METHOD PROTECTED ExecFaultHandling : BOOL
VAR
	bEnableCheck: BOOL ; // enable check functions 
	nActPos		: LREAL; // actual position of traverse axis (for readability)	 
	bActMovFwd	: BOOL ; // traverse is moving in positive direction
	bActMovRev	: BOOL ; // traverse is moving in negative direction
END_VAR
// ====== Write axis position to temporary variable to improver readability =======
	nActPos := stTraverseAxisRef.NcToPlc.ActPos ;
	IF stTraverseAxisRef.Status.Moving THEN 
		bActMovFwd := stTraverseAxisRef.Status.PositiveDirection ; 
		bActMovRev := stTraverseAxisRef.Status.NegativeDirection ; 
	ELSE
		bActMovFwd := FALSE ; 
		bActMovRev := FALSE ; 
	END_IF
	
// ====== Alway check if cylinder is down when within minimum range ======
	fbTimerStartup(IN := NOT bErrorActive, PT := LREAL_TO_TIME(stParTimeToClose.fValue));
	
	IF fbTimerStartup.Q 
	AND	nActPos > nTriggerPosUprev 
	AND nActPos < nTriggerPosUpFw 
	AND NOT fbSensorClosed.bFcoInputActive  THEN 	
		// Set error to active (stop traverse axis) 
		bErrorActive := TRUE ;
		// add message data
		stFault.Active			:= TRUE 								;
		stFault.Discription		:= 'support not in safe (down) position';
		stFault.MessageNumber	:= E_MessageNumbers.FF_Collision 		;
		stFault.FaultType		:= E_FaultTypes.FF				;
		refFbFault.CmdAddFault( stFault );
	END_IF

// ====== Make sure support Moves down ======
	IF bActMovFwd 
	AND nActPos > nTriggerPosCheckDownFw 
	AND nActPos < nTriggerPosUpFw 
	AND NOT fbSensorClosed.bFcoInputActive THEN 
		// Set error to active (stop traverse axis) 
		bErrorActive := TRUE ;
		// add message data
		stFault.Active			:= TRUE 								;
		stFault.Discription		:= 'Emergency stop support cylinder not down';
		stFault.MessageNumber	:= E_MessageNumbers.FF_Collision 		;
		stFault.FaultType		:= E_FaultTypes.FF				;
		refFbFault.CmdAddFault( stFault );
	ELSIF bActMovRev 
	AND nActPos > nTriggerPosUprev
	AND nActPos < nTriggerPosCheckDownRe 
	AND NOT fbSensorClosed.bFcoInputActive THEN 
		// Set error to active (stop traverse axis) 
		bErrorActive := TRUE ;
		// add message data
		stFault.Active			:= TRUE 								;
		stFault.Discription		:= 'Emergency stop support cylinder not down';
		stFault.MessageNumber	:= E_MessageNumbers.FF_Collision 		;
		stFault.FaultType		:= E_FaultTypes.FF				;
		refFbFault.CmdAddFault( stFault );
 	END_IF
END_METHOD

METHOD Init_Support : BOOL
VAR_INPUT
	sInValveName		: STRING			:= 'valve'	; // Name of the cylinder ( used for fault handling and identification)
	nInValveNumber		: UDINT				:= 0		; // Cylinder identification number
	// Support data
	nInSupportPosition	: LREAL := 0 		; // possition of support cylinder in reference to the home position 
	nInSupportWidth		: LREAL := 100		; // width of support cylinder 
	// Traverse data 
	nInTravMaxAcc			: LREAL ; // traverse maximum acceleration 
	nInTravMaxDec			: LREAL ; // traverse maximum deceleration 
	nInTraverseLength		: LREAL	:= 550		; // Length of sewing head cart 
	nInTraverseFlagPosition	: LREAL	:= 0		; // position of flag in reference to edge of cart 
	// cart data
	nInHandCartLenght		: LREAL := 250		; // hand cart length [mm]
	nInHandCartClearance	: LREAL := 300		; // Clearance around cart in which support is down

	// safety values 	
	nInMinSafeDistanceDown: LREAL := 200		; // Minimum distance for support to move down
	// Command state
	eResetState		: E_ValveResetState := 0		; // Cylinder reset state variable (default is idle) 
	eSafeState		: E_ValveResetState	:= 0		; // Valve safe state
END_VAR
// ====== initi valve ======
	SUPER^.Init(nInValveNumber, eResetState, eSafeState);
	
// ====== Set support data =======
	nSupportPosition 	:= nInSupportPosition 	;
	nSupportWidth		:= nInSupportWidth 		;

// ====== Set traverse Data ======
	nTravMaxAcc				:= nInTravMaxAcc			;
	nTravMaxDec				:= nInTravMaxDec			;
	nTraverseLength 		:= nInTraverseLength		;
	nTraverseFlagPosition	:= nInTraverseFlagPosition 	;
	nMinSafeDistanceDown	:= nInMinSafeDistanceDown	;

// ===== set handcart data =====
	nHandCartLength 		:= nInHandCartLenght 		;
	nHandCartClearance		:= nInHandCartClearance		;

// ====== set feedback to true (support always has feedback) =======
	bIcfFbkClosedPresent 	:= TRUE ;
	bIcfFbkOpenPresent		:= TRUE ;
	
// ====== Check if init is done ======
END_METHOD

METHOD PUBLIC Mod_ManualControl : BOOL
VAR_INPUT
	eCmdCylinder : E_CylinderCmd ; // cylinder manual command	
END_VAR
bCmdManual := TRUE ;

CASE eCmdCylinder OF
	E_CylinderCmd.Cyl_Reset:
		CmdReset();
	E_CylinderCmd.Cyl_Hold:
		CmdHold();
	E_CylinderCmd.Cyl_Teach:
		CmdTeach();
	E_CylinderCmd.Cyl_Calculate:
		ExecCalc();
	E_CylinderCmd.Cyl_Expand:
		CmdOpen();
	E_CylinderCmd.Cyl_Retract:
		CmdClose();
	ELSE 
		RETURN;
END_CASE
END_METHOD

METHOD Mod_SupportDown : BOOL
VAR_INPUT
END_VAR
bCmdSupportDown := true ;
END_METHOD

END_FUNCTION_BLOCK

// Axis/FunctionBlocks/FB_DevBasicACAxis
FUNCTION_BLOCK PUBLIC FB_DevBasicACAxis EXTENDS FB_DevBase
VAR_INPUT
	// ===== General Function input =====
		fCmdAcc			: LREAL := 15000;
		fCmdDecc		: LREAL := 15000; 
	// Manual control reference
		stManualCtrl	: UDT_ManualAxisCtrl ;
END_VAR
VAR_OUTPUT
	bHomed			: BOOL 	:= FALSE; 
	bMoving		: BOOL ; // Axis is moving
	bInPosition : BOOL ; // Axis is in position 
END_VAR
VAR
		AxisRef	: AXIS_REF ; // reference to AC axis
	// ===== HW Config Bits =====
		bIcfCmdVelocityRpm	: BOOL ; // input speeds in Rpm
		bIcfEnableForward 	: BOOL ; // Enable forward motion
 		bIcfEnablereverse	: BOOL ; // Enable reverse motion
		bIcfAlwaysEnable	: BOOL ; // 1 = Axis always enabled, 0 = Axis disabled at Idle 
		bIcfSimulationMode	: BOOL := FALSE ; // Simulation mode is active [default set to False] 
	// ===== Internal motion values ======
		fHomePosition		: LREAL := 0 ; // set position at homing
	// ====== Axis Settings ======
		fMaxVelo		: LREAL := 0 ; // Axis Maximum velocity
		fMaxAcc			: LREAL := 0 ; // Axis Maximum cceleration
		fMaxDec			: LREAL := 0 ; // axis Maxium deceleration 
		
		fSafeVeloLimit	: LREAL	:= 200; // Safe velocity limit 
		tEnableDelay	: TIME 	:= T#150MS	;
		tDisableDelay	: TIME 	:= T#500MS  ;
		
	// ====== Axis enable =====	
		bCmdEnableAxis 		: BOOL 	:= FALSE; // Command to enable the axis (External)
		bInternalEnable		: BOOL 	:= FALSE; // internal enable command (turns off after set time, and on at new motion command
		bDelayedEnable		: BOOL 	:= false; // Delayed enable signal for motion commands
		TonMotionEnable		: TON 			; // Timer on for motion command enable
		TofIntAxisEnable	: TOF  			; // Timer off for internal axis enable 
	// ===== Safe commands =====
		bCmdSafeStop	: BOOL ;
	// Motion commands 
		fbMcPower 			: MC_Power		;		// FB for enable and override
		fbMcReset 			: MC_Reset		;		// FB to reset axis
		fbSoeReset			: FB_SoEReset	; 		// FB to reset axis hardware
		fbMcHome			: MC_Home		;		// Fb to home Axis
		fbMcStop 			: MC_Stop		;		// FB to stop axis
		fbMcHalt			: MC_Halt		;		// FB to halt axis
		fbMcJog				: MC_Jog		;		// FB to Jog axis
		fbMcMoveVelocity	: MC_MoveVelocity;		// FB to move with specified velocity until Next command is given
	(* PtoP Motion move commands are in arrays so multiple commands can be stacked *) 
		fbMCMoveRelative	: ARRAY [0..1] OF MC_MoveRelative	;		// FB to move relative
		fbMcMoveAbsolute	: ARRAY [0..1] OF MC_MoveAbsolute	;		// FB to move axis (velocity movement)
		
	// Parameters 
		stMParMaxAcc : Udt_Parameter := (fMaximum := 999999, fMinimum := 0, fValue := 0)	; // Parameter for maximum acceleration
		stMParMaxDec : Udt_Parameter := (fMaximum := 999999, fMinimum := 0, fValue := 0)	; // Parameter for maximum Deceleration
		stMparMaxVelo: Udt_Parameter := (fMaximum := 999999, fMinimum := 0, fValue := 0)	; // Parameter for maximum velocity
		
	// Device feedback
		nActVelocity AT%I* : INT ; // actual speed of the motor
		nActPosition AT%I* : UDINT ; // Actual position of the motor

	// ===== Function execute triggers =====
		bExec_Reset			: BOOL := FALSE; // Execute reset
		bExec_Halt			: BOOL := FALSE; // Execute hold
		bExec_Home			: BOOL := FALSE; // Execute Home
		bExec_JogPositive	: BOOL := FALSE; // Execute Jog in positive direction
		bExec_JogNegative	: BOOL := FALSE; // Execute Jog in negative direction
		bExec_MoveVelocity	: BOOL := FALSE; // Execute move velocity
		arExec_MoveRelative	: ARRAY [0..1] OF BOOL ; // Execute move relative
		arExec_MoveAbs		: ARRAY [0..1] OF BOOL ; // Execute move absolute reverse
		

END_VAR

// Call base function
SUPER^(refFbFault := refFbFault);

// ==== Check if axis is initiated =====
IF NOT bInitOk THEN 
	RETURN ; 
END_IF

// ===== Execute safe functions =====
	ExecSafeFunctions(); 

// ==== Execute organizational functions =====
	ExecEnable();

// ==== execute motion functions =====
	CallMotionFunctions();

METHOD PUBLIC CmdHalt : BOOL
VAR_INPUT
	fDeceleration 	: LREAL := 0 ; // command deceleration
	mcBuffermode	: MC_BufferMode ; // Buffermode defines how the previous command is executed.
END_VAR
// Set command to true 
bExec_Halt 		:= TRUE ;
bInternalEnable	:= TRUE ;

// coppy parameters
fbMcHalt.Deceleration	:= fDeceleration;
fbMcHalt.BufferMode		:= mcBuffermode	;

// Set feedback output 
CmdHalt := fbMchalt.Active ;
END_METHOD

METHOD PUBLIC CmdHome : BOOL // start axis homing procedure
VAR_INPUT
	fPosition 		: LREAL := 0 ; // Homing position
	mcBufferMode	: MC_BufferMode := MC_BufferMode.MC_Aborting		; // Buffermode
END_VAR
// set command to true 
bExec_Home 		:= TRUE	; 
bInternalEnable	:= TRUE ;

// coppy parameters
fbMcHome.Position 	:= fPosition 	;
fbMcHome.BufferMode	:= mcBufferMode ;

// Set feedback output
CmdHome := fbMcHome.Done ;
END_METHOD

METHOD PUBLIC CmdJog : BOOL // Jog axis with variable speed. jog stops as soon as the command is false
VAR_INPUT
	fVelocity		: LREAL 	; // jog velocity can be adjusted as long as the command is active
	fPos			: LREAL 	; // Jog position or step size (if aplicable)
	bJogNegative 	: BOOL 		:= FALSE ; // jog in negative direction
	eJogmode		: E_JogMode := E_JogMode.MC_JOGMODE_CONTINOUS ; // jogmode [default MC_JOGMODE_CONTINOUS] 
END_VAR
// Velocity conversion from RPM to deg/sec
	IF bIcfCmdVelocityRpm THEN 
		fVelocity := Rpm_To_DegS(fVelocity);
	END_IF

// Set command to true
	IF fbMcJog.Velocity = fVelocity THEN // If command velocity changes, then set exec to false for one cycle to trigger new velocity so the jog follows the set velocity
		bExec_JogPositive	:= NOT bJogNegative ;
		bExec_JogNegative 	:= bJogNegative ;
	END_IF
	bInternalEnable			:= TRUE ;

// coppy parameters
	fbMcJog.Velocity	:= fVelocity 	;
	fbmcjog.Mode		:= eJogmode		;
	fbMcJog.Position	:= fPos			;

// Set feedback output 
	CmdJog := fbMcJog.Active ;
END_METHOD

METHOD PUBLIC CmdManual : BOOL
VAR
	eJogmode		: E_JogMode := E_JogMode.MC_JOGMODE_CONTINOUS ; // jogging mode 
END_VAR
// Enable axis for manual control
bCmdManual := TRUE ;

// set jog mode 
IF stManualCtrl.bCmdInching THEN 
	eJogmode := E_JogMode.MC_JOGMODE_INCHING ;
END_IF

// execute motion commands
IF stManualCtrl.bCmdJogForward OR stManualCtrl.bCmdJogReverse THEN 
	CmdJog (fVelocity := stManualCtrl.fVelocity, 
			fPos := stManualCtrl.fDistance, 
			bJogNegative := stManualCtrl.bCmdJogReverse, 
			eJogmode := eJogmode);
ELSIF stManualCtrl.bCmdToPos THEN 
	CmdMoveAbs( fPosition := stManualCtrl.fPosition, 
				fVelocity := stManualCtrl.fVelocity, 
				mcBuffermode := MC_BufferMode.MC_Aborting);
ELSIF stManualCtrl.bCmdHome THEN 
	CmdHome( fPosition := 0, mcBufferMode := MC_Aborting);
ELSE 
	CmdHalt( 	fDeceleration := fMaxDec * 0.9, 
				mcBuffermode := MC_BufferMode.MC_Aborting) ; 
END_IF
END_METHOD

METHOD PUBLIC CmdMoveAbs : BOOL // Move absolute command
VAR_INPUT
	fPosition	:	LREAL 	; // target position
	fVelocity	: 	LREAL 	; // Maximum velocity [units/sec]
	mcBuffermode: 	MC_BufferMode ; // Buffermode defines how the previous command is executed.
END_VAR
// Velocity conversion from RPM to deg/sec
	IF bIcfCmdVelocityRpm THEN 
		fVelocity := Rpm_To_DegS(fVelocity);
	END_IF

// Determine function for command stacking
	IF fbMcMoveAbsolute[0].Active THEN 
		arExec_MoveAbs[1] 				:= (fPosition <> fbMcMoveAbsolute[0].Position OR fVelocity <> fbMcMoveAbsolute[0].Velocity) ;
		fbMcMoveAbsolute[1].Position 	:= fPosition ;
		fbMcMoveAbsolute[1].Velocity 	:= fVelocity ; 
		fbMcMoveAbsolute[1].BufferMode 	:= mcBuffermode ;
	ELSE
		arExec_MoveAbs[0] 				:= (fPosition <> fbMcMoveAbsolute[1].Position OR fVelocity <> fbMcMoveAbsolute[1].Velocity) ;
		fbMcMoveAbsolute[0].Position 	:= fPosition ;
		fbMcMoveAbsolute[0].Velocity 	:= fVelocity ; 
		fbMcMoveAbsolute[0].BufferMode 	:= mcBuffermode ;
	END_IF

bInternalEnable	:= TRUE ;
// set feedback
IF arExec_MoveAbs[1] OR fbMcMoveAbsolute[1].Busy THEN 
	CmdMoveAbs :=	fbMcMoveAbsolute[1].Active ;
ELSE 
	CmdMoveAbs :=	fbMcMoveAbsolute[0].Active ;
END_IF
END_METHOD

METHOD CmdMoveRelative : BOOL // move relative command 
VAR_INPUT
	fDistance	:	LREAL 	; // target position
	fVelocity	: 	LREAL 	; // Maximum velocity [units/sec]
	mcBuffermode: 	MC_BufferMode ; // Buffermode defines how the previous command is executed.
END_VAR
// Velocity conversion from RPM to deg/sec
	IF bIcfCmdVelocityRpm THEN 
		fVelocity := Rpm_To_DegS(fVelocity);
	END_IF

// Determine function for command stacking
	IF fbMCMoveRelative[0].Active THEN 
		arExec_MoveRelative[1] := (fDistance <> fbMCMoveRelative[0].Distance OR fVelocity <> fbMCMoveRelative[0].Velocity) ;
		fbMCMoveRelative[1].Velocity	:= fVelocity 	;
		fbMCMoveRelative[1].Distance	:= fDistance	;
		fbMCMoveRelative[1].BufferMode	:= mcBuffermode	;
	ELSE 
		arExec_MoveRelative[0] := (fDistance <> fbMCMoveRelative[1].Distance OR fVelocity <> fbMCMoveRelative[1].Velocity) ;
		fbMCMoveRelative[0].Velocity	:= fVelocity 	;
		fbMCMoveRelative[0].Distance	:= fDistance	;
		fbMCMoveRelative[0].BufferMode	:= mcBuffermode	;
	END_IF

bInternalEnable	:= TRUE ;

// set feedback
IF arExec_MoveRelative[1] OR fbMCMoveRelative[1].Busy THEN 
	CmdMoveRelative :=	fbMCMoveRelative[1].Active ;
ELSE
	CmdMoveRelative :=	fbMCMoveRelative[0].Active ;
END_IF
END_METHOD

METHOD PUBLIC CmdMoveVelocity : BOOL // Move with set velocity until stopped
VAR_INPUT
	fVelocity	: 	LREAL 	; // Maximum velocity [units/sec]
	mcDirection : 	MC_Direction := MC_Direction.MC_Positive_Direction ; // Direction of movement mc_direction [ deafult mc_positive_direction]
	mcBuffermode: 	MC_BufferMode ; // Buffermode defines how the previous command is executed.
END_VAR
// Velocity conversion from RPM to deg/sec
	IF bIcfCmdVelocityRpm THEN 
		fVelocity := Rpm_To_DegS(fVelocity);
	END_IF

// Set command to true 
	bExec_MoveVelocity 	:= TRUE ;
	bInternalEnable		:= TRUE ;

// coppy parameters
	fbMcMoveVelocity.Velocity	:= fVelocity 	;
	fbMcMoveVelocity.Direction 	:= mcDirection	;
	fbMcMoveVelocity.BufferMode	:= mcBuffermode	;

// Set feedback output 
	CmdMoveVelocity := fbMcMoveVelocity.Active ;
END_METHOD

METHOD PUBLIC CmdReset : BOOL
VAR_INPUT
END_VAR
// Set reset axis to true 				
	bExec_Reset 	:= TRUE ; 
	bInternalEnable	:= TRUE ;
	
// Set feedback output 
	CmdReset := fbMcReset.Done ;
END_METHOD

METHOD PUBLIC CmdSafeStop : BOOL
VAR_INPUT
END_VAR
// Set safestop command
bCmdSafeStop := TRUE ; 

// Set feedback output 
CmdSafeStop := bDevIsSafe OR NOT bInitOk;
END_METHOD

METHOD PUBLIC Init : BOOL
VAR_INPUT
	// Axis message Data 
	nDevNumber	: UDINT		:= 0	; // Axis number 
	// Config Bits
	bIcfCmdVelocityRpm	: BOOL := FALSE ; // input speeds in Rpm
	bIcfEnableForward 	: BOOL := TRUE 	; // Enable forward motion
	bIcfEnablereverse	: BOOL := TRUE 	; // Enable reverse motion
	bIcfAlwaysEnable	: BOOL := FALSE ; // 1 = Axis always enabled, 0 = Axis disabled at Idle 
	bIcfSimulationMode	: BOOL := FALSE ; // Simulation mode is active [default set to False] Used for testing without hardware present 
	
	fHomePosition		: LREAL := 0 	; // set position at homing
	fSafeVeloLimit		: LREAL	:= 360 	; // safe velocity limit [deg/sec]
	nEncTurnoverVal 	: LREAL := 360	; // encoder turnover value 
	tEnableDelay		: time 	:= T#0MS; // Time between axis enable command and motion command execution (0 := no delay active)	
	tDisabledelay		: TIME 	:= T#100MS; // Axis idle time before axis is disabled 
END_VAR
VAR 
	bActParamValid 		: BOOL ; // Parameter read is valid 
END_VAR
// Calculate device number
	THIS^.nDevNumber := nDevNumber ;
	SUPER^.CalcDeviceId();

// ===== Message data set =====
	stFault.ComponentType		:= E_ComponentTypes.Axis ;
	
// ===== Write parameters =====
	stMParMaxAcc.nNumber		:= nDevId + 1;
	stMParMaxAcc.sDiscription 	:= CONCAT(STR1 := sDevName, STR2:= ' hardware maximum accaleration (0 = HWMaximum)'); 
	stMParMaxAcc.sName			:= CONCAT(STR1 := sDevName, STR2:= 'HardMaxAceleration');
	stMParMaxAcc.sType			:= 'MPar';
	stMParMaxAcc.sUnit			:= 'Units/Sec^2';
	
	stMParMaxDec.nNumber		:= nDevId + 2;
	stMParMaxDec.sDiscription 	:= CONCAT(STR1 := sDevName, STR2:= ' hardware maximum deceleration(0 = HWMaximum)'); 
	stMParMaxDec.sName			:= CONCAT(STR1 := sDevName, STR2:= 'HardMaxDeceleration');
	stMParMaxDec.sType			:= 'MPar';
	stMParMaxDec.sUnit			:= 'Units/Sec^2';
	
	stMparMaxVelo.nNumber		:= nDevId + 3;
	stMparMaxVelo.sDiscription 	:= CONCAT(STR1 := sDevName, STR2:= ' hardware maximum velocity'); 
	stMparMaxVelo.sName			:= CONCAT(STR1 := sDevName, STR2:= 'HardMaxVelocity');
	stMparMaxVelo.sType			:= 'MPar';
	stMparMaxVelo.sUnit			:= 'Units/Sec';

	refFbParHandler.CmdAddParameter(refParameter := stMParMaxAcc);
	refFbParHandler.CmdAddParameter(refParameter := stMParMaxDec);
	refFbParHandler.CmdAddParameter(refParameter := stMparMaxVelo);

// ===== set axis configuration =====	
	fMaxAcc	:= stMParMaxAcc.fValue;
	fMaxDec	:= stMParMaxDec.fValue;	
	fMaxVelo:= stMparMaxVelo.fValue;

	fCmdAcc 		:= fMaxAcc;
	fCmdDecc		:= fMaxDec;
// ===== Configure Axis =====
	// ***** Config Bits *****
		THIS^.bIcfCmdVelocityRpm	:= bIcfCmdVelocityRpm	; // Enable speed inputs in Rpm
		THIS^.bIcfEnableForward 	:= bIcfEnableForward 	; // Enable forward motion
		THIS^.bIcfEnablereverse		:= bIcfEnablereverse	; // Enable reverse motion
		THIS^.bIcfAlwaysEnable		:= bIcfAlwaysEnable		; // Always enable motor and brake if safety is ok
		THIS^.bIcfSimulationMode	:= bIcfSimulationMode 	; // Simulation mode is active [default set to False] 

	// ***** config homing Mode ***** 
 		THIS^.fHomePosition			:= fHomePosition;
	// ***** Velocity settings *****
		THIS^.fSafeVeloLimit 		:= fSafeVeloLimit ; // set maximum safe velocity	
	// ***** Time delay enable off *****
		THIS^.tEnableDelay		:= tEnableDelay	;
		THIS^.tDisableDelay 	:= tDisabledelay ;		

// ===== Set device type for manual control =====
	eDevType := E_Devices.Axis ;
		
// ===== reset axis state indicators ======
	bErrorActive 	:= FALSE;

// ====== Set init to done =======
	bInitOk	:= TRUE ;
END_METHOD

METHOD PRIVATE ExecEnable : BOOL
VAR_INPUT
END_VAR
// ===== Set axis enable ======
IF NOT bEnable AND NOT bCmdManual AND nActVelocity <> 0 THEN
	CmdHalt(fDeceleration := fCmdDecc, mcBuffermode := MC_BufferMode.MC_Aborting);
ELSE 
	bCmdEnableAxis	:= bEnable OR bCmdManual ;
	bCmdManual := FALSE ;
END_IF

// ===== Check if axis is bussy with a command =====
	bInternalEnable	S= bIcfAlwaysEnable ; // always enable axis if configured
	
// ===== Axis disable timer after last command =====
	TofIntAxisEnable (	IN:= bInternalEnable, PT := tDisableDelay);

// ===== Enable drive =====
	fbMcPower(	Axis			:= AxisRef , 
				Enable			:= bCmdEnableAxis AND TofIntAxisEnable.Q, 
				Enable_Positive	:= bIcfEnableForward, 
				Enable_Negative	:= bIcfEnablereverse, 
				Override		:= 100 );  
				
// ===== Reset internal enable signal =====
	bInternalEnable := FALSE ; 	

// ===== Delayed enable function =====	
	TonMotionEnable(IN := fbMcPower.Active, PT := tEnableDelay);
	bDelayedEnable := TonMotionEnable.Q ;	


IF fbMcPower.Error THEN 
	bErrorActive			:= TRUE							;
	stFault.Active 			:= TRUE 						;
	stFault.MessageNumber	:= E_MessageNumbers.FF_AxisFault;
	stFault.Discription		:= CONCAT('Enable Fault ', UDINT_TO_STRING(fbMcPower.ErrorID));				;
	stFault.FaultType		:= E_FaultTypes.FF				;
	refFbFault.CmdAddFault( stFault );
END_IF
END_METHOD

METHOD PRIVATE ExecHalt : BOOL
VAR_INPUT
END_VAR
// ==== Execute halt function ===== 
fbMcHalt (	Axis 		:= AxisRef,
			Execute 	:= bExec_Halt );

// ===== reset command =====
	bExec_Halt := FALSE ;
	bInternalEnable := fbMcHalt.Busy ;			
	
// Halt fault handling 
	IF fbMcHalt.Error THEN 
		bErrorActive			:= TRUE							;
		stFault.Active 			:= TRUE 						;
		stFault.MessageNumber	:= E_MessageNumbers.FF_AxisFault;
		stFault.Discription		:= CONCAT('Halt Fault ', UDINT_TO_STRING(fbMcHalt.ErrorID));				;
		stFault.FaultType		:= E_FaultTypes.FF				;
		refFbFault.CmdAddFault( stFault );
	END_IF
END_METHOD

METHOD PRIVATE ExecHome : BOOL
VAR_INPUT
END_VAR
// ==== execute homing function =====
	fbMcHome(	Axis			:= AxisRef,
				Execute			:= bExec_Home,
				HomingMode		:= MC_DefaultHoming ); 
			
// Reset exec command 
	bExec_Home 	:= FALSE ;
	bHomed		S= fbMcHome.Done ;	
	bInternalEnable := fbMcHome.Busy ;			
				
// fault handling 
	IF fbMcHome.Error THEN 
		bErrorActive			:= TRUE							;
		stFault.Active 			:= TRUE 						;
		stFault.MessageNumber	:= E_MessageNumbers.FF_AxisFault;
		stFault.Discription		:= CONCAT('Homing Fault ', UDINT_TO_STRING(fbMcHome.ErrorID));				;
		stFault.FaultType		:= E_FaultTypes.FF				;
		refFbFault.CmdAddFault( stFault );
	END_IF
END_METHOD

METHOD PRIVATE ExecJog : BOOL
VAR_INPUT
END_VAR
// ===== Execute Jog function =====
	// function call
	fbMcJog (	Axis 		:= AxisRef,
				JogForward	:= bExec_JogPositive,
				JogBackwards:= bExec_JogNegative,
				Acceleration:= fCmdAcc,
				Deceleration:= fCmdDecc );

// ===== reset command =====
	bExec_JogPositive 	:= FALSE  ;
	bExec_JogNegative	:= FALSE  ;
	bInternalEnable		:= fbMcJog.Busy; 

// Jog fault handling 
	IF fbMcJog.Error THEN 
		bErrorActive			:= TRUE							;
		stFault.Active 			:= TRUE 						;
		stFault.MessageNumber	:= E_MessageNumbers.FF_AxisFault;
		stFault.Discription		:= CONCAT('Jog Fault ', UDINT_TO_STRING(fbMcJog.ErrorID));				;
		stFault.FaultType		:= E_FaultTypes.FF				;
		refFbFault.CmdAddFault( stFault );
	END_IF
END_METHOD

METHOD PRIVATE ExecMoveAbsolute : BOOL
VAR_INPUT
END_VAR
VAR
	i : UDINT := 0 ;
END_VAR
// ==== execute move absolute function =====
FOR i := 0 TO 1 DO 
	// function call
	fbMcMoveAbsolute[i](	Axis 		:= AxisRef,
							Execute 	:= arExec_MoveAbs[i],
							Acceleration:= fCmdAcc,
							Deceleration:= fCmdDecc );  
	// reset Exec command 
	arExec_MoveAbs[i] := FALSE ; 
	bInternalEnable := fbMcMoveAbsolute[i].Busy ;			

	// If function is done then reset command values
	IF fbMcMoveAbsolute[i].Done THEN 
		fbMcMoveAbsolute[i].Velocity	:= 0 ;
		fbMcMoveAbsolute[i].Position	:= 0 ; 
	END_IF
	
	// fault handling 
	IF fbMcMoveAbsolute[i].Error THEN 
		bErrorActive			:= TRUE							;
		stFault.Active 			:= TRUE 						;
		stFault.MessageNumber	:= E_MessageNumbers.FF_AxisFault;
		stFault.Discription		:= CONCAT('Move absolute Fault ', UDINT_TO_STRING(fbMcMoveAbsolute[i].ErrorID));				;
		stFault.FaultType		:= E_FaultTypes.FF				;
		refFbFault.CmdAddFault( stFault );
	END_IF
END_FOR
END_METHOD

METHOD PRIVATE ExecMoveRelative : BOOL
VAR_INPUT
END_VAR
VAR
	i : UDINT := 0 ;
END_VAR
// ===== Execute move relative function ======
FOR i := 0 TO 1 DO 
	// function call
	fbMCMoveRelative[i](	Axis 		:= AxisRef,
							Execute		:= arExec_MoveRelative[i],
							Acceleration:= fCmdAcc,
							Deceleration:= fCmdDecc );
	// reset Exec command 
	arExec_MoveRelative[i] := FALSE ; 
	bInternalEnable := fbMCMoveRelative[i].Busy ;			

	// If function is done then reset command values
	IF fbMCMoveRelative[i].Done THEN 
		fbMCMoveRelative[i].Velocity	:= 0 ;
		fbMCMoveRelative[i].Distance	:= 0 ; 
	END_IF
	
	// fault handling 
	IF fbMCMoveRelative[i].Error THEN 
		bErrorActive			:= TRUE							;
		stFault.Active 			:= TRUE 						;
		stFault.MessageNumber	:= E_MessageNumbers.FF_AxisFault;
		stFault.Discription		:= CONCAT('Move relative Fault ', UDINT_TO_STRING(fbMCMoveRelative[i].ErrorID));				;
		stFault.FaultType		:= E_FaultTypes.FF			;
		refFbFault.CmdAddFault( stFault );
	END_IF
END_FOR
END_METHOD

METHOD PRIVATE ExecMoveVelocity : BOOL
VAR_INPUT
END_VAR
// ===== Execute move velocity function =====
// function call
fbMcMoveVelocity (	Axis 		:= AxisRef,
					Execute		:= bExec_MoveVelocity,
					Acceleration:= fCmdAcc,
					Deceleration:= fCmdDecc );

// ===== reset command =====
bExec_MoveVelocity := FALSE ;
bInternalEnable		:= fbMcMoveVelocity.Busy;
	
// Halt fault handling 
IF fbMcHalt.Error THEN 
	bErrorActive			:= TRUE							;
	stFault.Active 			:= TRUE 						;
	stFault.MessageNumber	:= E_MessageNumbers.FF_AxisFault;
	stFault.Discription		:= CONCAT('Move velocity Fault ', UDINT_TO_STRING(fbMcMoveVelocity.ErrorID));				;
	stFault.FaultType		:= E_FaultTypes.FF				;
	refFbFault.CmdAddFault( stFault );
END_IF
END_METHOD

METHOD PRIVATE ExecReset : BOOL
VAR_INPUT
END_VAR
IF  nActVelocity <> 0 AND bExec_Reset THEN // If the axis is still moving execute safe stop first
	CmdSafeStop();
	RETURN;
END_IF

// perform reset 
	fbMcReset	( 	Execute	:= bexec_reset AND NOT fbSoeReset.Busy,
					Axis	:= AxisRef ); 
					
// ===== reset command =====
	bExec_Reset := FALSE ;
	
// ===== reset internal fault bits and stop bits =====
	bErrorActive 			:= FALSE ; 
	
// ===== reset safe commands ======
	bCmdSafeStop	:= FALSE ; 
	
// Reset fault handling 
	IF fbSoeReset.Error OR fbMcReset.Error THEN 
		bErrorActive			:= TRUE							;
		stFault.Active 			:= TRUE 						;
		stFault.MessageNumber	:= E_MessageNumbers.FF_AxisFault;
		stFault.Discription		:= CONCAT('Reset Fault ', UDINT_TO_STRING(fbMcReset.ErrorID))			;
		stFault.FaultType		:= E_FaultTypes.FF				;
		refFbFault.CmdAddFault( stFault );
	END_IF
END_METHOD

METHOD PRIVATE ExecSafeFunctions : BOOL
VAR_INPUT
END_VAR
// ==== Stop when safety is not ok =====
	bCmdSafeStop := NOT bSafetyOk ;

// ==== Safe operation functions (overrule all other motion functions) =====
	fbMcStop( 	Axis 			:= AxisRef		,
				Execute 		:= bCmdSafeStop	,
				Deceleration	:= fMaxDec		);
	
	// Reset axis command			
	bCmdSafeStop 	R= fbMcStop.Done ;
	
// Safestop fault handling 
	IF fbMcStop.Error THEN 
		bErrorActive			:= TRUE							;
		stFault.Active 			:= TRUE 						;
		stFault.MessageNumber	:= E_MessageNumbers.FF_AxisFault;
		stFault.Discription		:= CONCAT('Safe stop axis fault ', UDINT_TO_STRING(fbMcStop.ErrorID));				;
		stFault.FaultType		:= E_FaultTypes.FF				;
		refFbFault.CmdAddFault( stFault );
	END_IF

// ===== Dev is safe feedback =====
bDevIsSafe := NOT bCmdEnableAxis  ;
END_METHOD

METHOD PRIVATE CallMotionFunctions : BOOL
VAR_INPUT
END_VAR
// ===== Check if safe to move =====
	IF bCmdSafeStop OR NOT bDelayedEnable THEN 
		RETURN ;
	END_IF

// ===== Homing functions =====
	ExecHome		(); 

// ===== Motion standstil commands =====
	ExecHalt		();

// ===== Motion move functions
	ExecJog			(); 
	ExecMoveAbsolute();
	ExecMoveRelative();
	ExecMoveVelocity();
END_METHOD

END_FUNCTION_BLOCK

// Axis/FunctionBlocks/FB_DevHybridAc
FUNCTION_BLOCK PUBLIC FB_DevHybridAc EXTENDS Fb_DevAxis
VAR_INPUT
END_VAR
VAR_OUTPUT
END_VAR
VAR
	// Parameters 
		stMParMaxAcc : Udt_Parameter := (fMaximum := 999999, fMinimum := 0, fValue := 0)	; // Parameter for maximum acceleration
		stMParMaxDec : Udt_Parameter := (fMaximum := 999999, fMinimum := 0, fValue := 0)	; // Parameter for maximum Deceleration
		stMparMaxVelo: Udt_Parameter := (fMaximum := 999999, fMinimum := 0, fValue := 0)	; // Parameter for maximum velocity
END_VAR

SUPER^();

METHOD INTERNAL ExecHalt : BOOL
VAR_INPUT
END_VAR
// The hybrid axis is equiped with it's own safety stop system therefore mc halt is no longer needed with an Estop
IF bSafetyOk THEN 
	// ==== Execute halt function ===== 
	fbMcHalt (	Axis 		:= AxisRef,
				Execute 	:= bExec_Halt );
END_IF
// ===== reset command =====
	bExec_Halt := FALSE ;
	
// Halt fault handling 
	IF fbMcHalt.Error THEN 
		bError					:= TRUE							;
		stFault.Active 			:= TRUE 						;
		stFault.MessageNumber	:= E_MessageNumbers.FF_AxisFault;
		stFault.Discription		:= CONCAT('Halt Fault ', UDINT_TO_STRING(fbMcHalt.ErrorID));				;
		stFault.FaultType		:= E_FaultTypes.FF				;
		refFbFault.CmdAddFault( stFault );
	END_IF
END_METHOD

METHOD INTERNAL ExecReadStatus : BOOL
VAR_INPUT
END_VAR
// Read axis status from drive
AxisRef.ReadStatus();						
// convert velocity to RPM for output if aplicable
IF bIcfCmdVelocityRpm THEN 
	fVelocity := AxisRef.NcToPlc.ActVelo / 6 ;
ELSE 
	fVelocity := AxisRef.NcToPlc.ActVelo ;
END_IF

// write position output
fActPosition := AxisRef.NcToPlc.ActPos ;
						
// set status bits 
bIdle := NOT AxisRef.Status.HasJob ;
END_METHOD

METHOD INTERNAL ExecReset : BOOL
VAR_INPUT
END_VAR
IF  AxisRef.Status.Moving AND bExec_Reset THEN // If the axis is still moving execute safe stop first
	CmdSafeStop();
	RETURN;
END_IF

	fbMcReset	( 	Execute	:= bexec_reset,
					Axis	:= AxisRef ); 
					
// ===== reset command =====
	bExec_Reset := FALSE ;
	
// ===== reset internal fault bits and stop bits =====
	bError 			:= FALSE ; 
	
// ===== reset safe commands ======
	bCmdSafeStop	:= FALSE ; 
	bCmdSafeSpeed 	:= FALSE ;
	
// Reset fault handling 
	IF fbMcReset.Error THEN 
		bError					:= TRUE							;
		stFault.Active 			:= TRUE 						;
		stFault.MessageNumber	:= E_MessageNumbers.FF_AxisFault;
		stFault.Discription		:= CONCAT('Reset Fault ', UDINT_TO_STRING(fbMcReset.ErrorID))			;
		stFault.FaultType		:= E_FaultTypes.FF				;
		refFbFault.CmdAddFault( stFault );
	END_IF
END_METHOD

METHOD PUBLIC Init : BOOL
VAR_INPUT
	// Axis message Data 
	nDevNumber	: UDINT		:= 0	; // Axis number 
	// Config Bits
	bIcfCmdVelocityRpm	: BOOL := FALSE ; // input speeds in Rpm
	bIcfEnableForward 	: BOOL := TRUE 	; // Enable forward motion
	bIcfEnablereverse	: BOOL := TRUE 	; // Enable reverse motion
	bIcfAlwaysEnable	: BOOL := FALSE ; // 1 = Axis always enabled, 0 = Axis disabled at Idle 
	bIcfSimulationMode	: BOOL := FALSE ; // Simulation mode is active [default set to False] Used for testing without hardware present 
	
	// Config Values 
	mcHomingMode 		: MC_HomingMode := MC_HomingMode.MC_DefaultHoming; 
	fHomePosition		: LREAL := 0 	; // set position at homing
	fSafeVeloLimit		: LREAL	:= 360 	; // safe velocity limit [deg/sec]
	nEncTurnoverVal 	: LREAL := 360	; // encoder turnover value 
	tEnableDelay		: time 	:= T#0MS; // Time between axis enable command and motion command execution (0 := no delay active)	
	tDisabledelay		: TIME 	:= T#100MS; // Axis idle time before axis is disabled 
END_VAR
VAR 
	bActVeloReadValid 	: BOOL ; // velocity parameter read is valid 
	bActAccReadValid 	: BOOL ; // Acceleration parameter read is valid 
	bActDecReadValid 	: BOOL ; // Deceleration parameter read is valid 
	bActParamValid 		: BOOL ; // Parameter read is valid 
END_VAR
// Calculate device number
	THIS^.nDevNumber := nDevNumber ;
	SUPER^.CalcDeviceId();

// ===== Message data set =====
	stFault.ComponentType		:= E_ComponentTypes.Axis ;
	
// ===== Write parameters =====
	stMParMaxAcc.nNumber		:= nDevId + 1;
	stMParMaxAcc.sDiscription 	:= CONCAT(STR1 := sDevName, STR2:= ' hardware maximum accaleration (0 = HWMaximum)'); 
	stMParMaxAcc.sName			:= CONCAT(STR1 := sDevName, STR2:= 'HardMaxAceleration');
	stMParMaxAcc.sType			:= 'MPar';
	stMParMaxAcc.sUnit			:= 'Units/Sec^2';
	
	stMParMaxDec.nNumber		:= nDevId + 2;
	stMParMaxDec.sDiscription 	:= CONCAT(STR1 := sDevName, STR2:= ' hardware maximum deceleration(0 = HWMaximum)'); 
	stMParMaxDec.sName			:= CONCAT(STR1 := sDevName, STR2:= 'HardMaxDeceleration');
	stMParMaxDec.sType			:= 'MPar';
	stMParMaxDec.sUnit			:= 'Units/Sec^2';
	
	stMparMaxVelo.nNumber		:= nDevId + 3;
	stMparMaxVelo.sDiscription 	:= CONCAT(STR1 := sDevName, STR2:= ' hardware maximum velocity'); 
	stMparMaxVelo.sName			:= CONCAT(STR1 := sDevName, STR2:= 'HardMaxVelocity');
	stMparMaxVelo.sType			:= 'MPar';
	stMparMaxVelo.sUnit			:= 'Units/Sec';

	refFbParHandler.CmdAddParameter(refParameter := stMParMaxAcc);
	refFbParHandler.CmdAddParameter(refParameter := stMParMaxDec);
	refFbParHandler.CmdAddParameter(refParameter := stMparMaxVelo);

// ===== set axis configuration =====	
	fMaxAcc	:= stMParMaxAcc.fValue;
	fMaxDec	:= stMParMaxDec.fValue;	
	fMaxVelo:= stMparMaxVelo.fValue;

	fCmdAcc 		:= fMaxAcc;
	fCmdDecc		:= fMaxDec;
// ===== Configure Axis =====
	// ***** Config Bits *****
		THIS^.bIcfCmdVelocityRpm	:= bIcfCmdVelocityRpm	; // Enable speed inputs in Rpm
		THIS^.bIcfEnableForward 	:= bIcfEnableForward 	; // Enable forward motion
		THIS^.bIcfEnablereverse		:= bIcfEnablereverse	; // Enable reverse motion
		THIS^.bIcfAlwaysEnable		:= bIcfAlwaysEnable		; // Always enable motor and brake if safety is ok
		THIS^.bIcfSimulationMode	:= bIcfSimulationMode 	; // Simulation mode is active [default set to False] 

	// ***** config homing Mode ***** 
 		THIS^.mcHomingMode 			:= mcHomingMode ; // set homing mode
 		THIS^.fHomePosition			:= fHomePosition;
	// ***** Velocity settings *****
		THIS^.fSafeVeloLimit 		:= fSafeVeloLimit ; // set maximum safe velocity	
	// ***** Time delay enable off *****
		THIS^.tEnableDelay		:= tEnableDelay	;
		THIS^.tDisableDelay 	:= tDisabledelay ;		

// ===== Set device type for manual control =====
	eDevType := E_Devices.Axis ;
		
// ===== reset axis state indicators ======
	bErrorActive 	:= FALSE;

// ====== Set init to done =======
	bInitOk	:= TRUE ;
END_METHOD

END_FUNCTION_BLOCK

// Buttons/Functions/FB_DevHMIButton
FUNCTION_BLOCK PUBLIC FB_DevHMIButton EXTENDS FB_DevBase // Button function for HMI 
VAR_INPUT
	Istatus			: BOOL	:= FALSE;// Digital sensor, Direct input status
	tDelay			: TIME 	:= T#5S	;// Time before delayed signal becomes active 
END_VAR
VAR_OUTPUT
	bFcoInputActive		: BOOL 			;// Digital sensor, Button active state
	bFcoDelay			: BOOL			;// Button, Delayed input status (3 seconds) 
	bFeStatus			: BOOL			;// Button, Falling edge of input signal	
	bReStatus			: BOOL			;// Button, Rising edge of input signal
	TetInputActive		: TIME			;// Button, Time elapsed while button is active
	bInvisible			: BOOL 			;// Button, Button is made invisible
	bDeactivate			: BOOL 			;// Button, Deactivate button 
END_VAR
VAR
	FB_delIStatus: TON; // Timer function for delayed input status 
	FB_feIStatus: F_TRIG; // generate falling edge pulse edge from Istatus
	FB_reIStatus: R_TRIG; // generate falling edge pulse edge from Istatus
END_VAR

// Call base function
SUPER^();

// ***** Direct input when enabled *****
IF bEnable THEN 
	bFcoInputActive := Istatus ;
ELSE 
	bFcoInputActive := FALSE ;
END_IF

// ===== check if function is enabled =====
	IF NOT bEnable THEN 
		bInvisible 	:= TRUE ;
		bDeactivate	:= TRUE ;
		bFcoDelay	:= FALSE;
		RETURN;
	ELSE  
		bInvisible 	:= FALSE ;
		bDeactivate	:= FALSE ;
	END_IF

// ====== process functions if enabled ======
	// ***** Set Delayed inputs and time elapsed ****
		FB_delIStatus(	IN:= bFcoInputActive,
						PT:= tDelay , 
						Q=> bFcoDelay , 
						ET=> TetInputActive 
					  ); // Generate delayed input status from push button input status
	// ***** Edge triggers *****
		FB_feIStatus(CLK:= Istatus , Q=> bFeStatus ); // generate falling edge pulse on pushbutton input
		FB_reIStatus (Clk := Istatus , Q => bReStatus); // Generate rising edge from push button input signal

END_FUNCTION_BLOCK

// Buttons/Functions/FB_DevPushButton
FUNCTION_BLOCK PUBLIC FB_DevPushButton EXTENDS Fb_DevDigitalInputFunctions
VAR_INPUT
END_VAR
VAR_OUTPUT
END_VAR
VAR
END_VAR

// set device type
IF eDevType = E_Devices.Undefined THEN 
	eDevType := E_Devices.DigitalSensor ;
END_IF

SUPER^();

END_FUNCTION_BLOCK

// Encoders/FunctionBlocks/FB_EncoderBase
FUNCTION_BLOCK PUBLIC FB_EncoderBase
VAR_INPUT
	nCfgUnitsPerPulse	: LREAL := 1	; // Scale factor for output [units/pulse]
	nCfgOffset			: LREAL := 0	; // Offset for output
	
	bIcfInverted		: BOOL	:= FALSE; // Invert output position = standard false  
END_VAR
VAR_OUTPUT
	nOutPosition		: LREAL	:= 0	; // Scaled position output
	nOutRaw				: UDINT := 0	; // Raw output value	 
	nVelocity			: LREAL	:= 0 	; // Velocity [units/sec]
END_VAR
VAR
END_VAR

METHOD PUBLIC FastTask : BOOL
VAR_INPUT
END_VAR
END_METHOD

END_FUNCTION_BLOCK

// Encoders/FunctionBlocks/FB_EncoderInput
FUNCTION_BLOCK FB_EncoderInput EXTENDS FB_EncoderBase
VAR_INPUT
END_VAR
VAR_OUTPUT
END_VAR
VAR
	iEncoderSignal AT%I*: UDINT ;
	
	nScaledValue		: LREAL ; // Only scaled value for internal use
	nValueWithOffset	: LREAL ; // scaled value with added offset
END_VAR

// ====== Scale Output value ======
	nScaledValue := UDINT_TO_LREAL(iEncoderSignal) * nCfgUnitsPerPulse ;

// ====== Invert ======
	IF bIcfInverted THEN 
		nScaledValue := nScaledValue * -1;
	END_IF
	
// ====== Add offset ======= 
	nValueWithOffset := nScaledValue + nCfgOffset ;

// ====== Set Outputs =======
	nOutPosition 	:= nValueWithOffset ;
	nOutRaw			:= iEncoderSignal	;

METHOD PUBLIC FastTask : BOOL
VAR_INPUT
END_VAR
END_METHOD

END_FUNCTION_BLOCK

// HardwareDiagnostics/FB_ELModuleDiag
FUNCTION_BLOCK PUBLIC FB_ELModuleDiag
VAR_INPUT
END_VAR
VAR_OUTPUT
	bError 	:	BOOL ; // Module is in error
	sErrorDiscription : STRING ; // module error discription 
END_VAR
VAR
END_VAR

END_FUNCTION_BLOCK

// Outputs/AnalogOutputs/FB_DevAnalogOutputScaled
FUNCTION_BLOCK FB_DevAnalogOutputScaled EXTENDS FB_DevAnalogOutput
VAR_INPUT
END_VAR
VAR_OUTPUT
END_VAR
VAR
	fGainFactor 	: LREAL:= 32767	;
END_VAR

SUPER^();

METHOD INTERNAL ExecSetFeedback : BOOL
VAR_INPUT
END_VAR
// Set feedback 
fOutputValue := qnHwOut ;
END_METHOD

METHOD INTERNAL ExecSetOutput : BOOL
VAR_INPUT
END_VAR
// Set Output to physical device
IF bEnable OR bCmdManual THEN 
	qnHwOut := LREAL_TO_INT(fCmdValue * fGainFactor) ;
	qnHwOut := LIMIT(nLimitMin, qnHwOut, nLimitMax) ; 
ELSE 
	fCmdValue := 0 ; 
END_IF
END_METHOD

METHOD PUBLIC SetScaling : BOOL 
VAR_INPUT
	fMaxValue	: LREAL ; 		// Maximum input value after scaling, e.g. 100% (mandatory input)  
END_VAR
// calculate gain 
fGainFactor := nLimitMax / fMaxValue ;
END_METHOD

END_FUNCTION_BLOCK

// Sensors/AnalogInput/FunctionBlocks/FB_DevAnalogInAutoCalibrate
FUNCTION_BLOCK PUBLIC FB_DevAnalogInAutoCalibrate EXTENDS FB_DevAnalogInputScaled
VAR_INPUT
END_VAR
VAR_OUTPUT
END_VAR
VAR
END_VAR

SUPER^();

METHOD PUBLIC CmdCalibrateNull : BOOL
VAR_INPUT
END_VAR
// set offset to calibrate to null
nOfset := - inHwInput ;
END_METHOD

METHOD PUBLIC CmdCalilbrateValue : BOOL // calibrate gain factor to actual value (warning calibrate to null before calibrating to value)
VAR_INPUT
	fCalibrationValue	: LREAL ; // Active input value to sensor (calibration setpoint)
END_VAR
// set gain from current value
fGainFactor := INT_TO_LREAL(inHwInput + nOfset) / fCalibrationValue ;
END_METHOD

END_FUNCTION_BLOCK

// Sensors/AnalogInput/FunctionBlocks/FB_DevAnalogInputScaled
FUNCTION_BLOCK PUBLIC FB_DevAnalogInputScaled EXTENDS FB_DevAnalogInput
VAR_INPUT
END_VAR
VAR_OUTPUT
END_VAR
VAR
	fGainFactor 	: LREAL	:= 1	;
	nOfset			: INT	:= 0	;
END_VAR

SUPER^();

METHOD ExecSetFeedback : BOOL
VAR
	nCalibValue	: INT ; 
END_VAR
// Offset 
IF bCmdSimulate THEN 
	nCalibValue := fSimValue + nOfset ;
ELSE
	nCalibValue := inHwInput + nOfset ;
END_IF

fValue := INT_TO_LREAL(nCalibValue) / fGainFactor;
END_METHOD

METHOD PUBLIC SetScaling : BOOL 
VAR_INPUT
	fMaxValue	: LREAL ; 	// Maximum input value after scaling, e.g. 100%, 0 = no scaling (gain = hardware limit / fMaxValue)  
	fOfset		: LREAL ;	// offset value (fvalue = (gain * hwvalue) + fOfset)
END_VAR
// calculate gain 
IF fMaxValue =0 THEN 
	fGainFactor := 1 ;
ELSE 
	fGainFactor := nLimitMax / fMaxValue ;
END_IF

nOfset := LREAL_TO_INT(fOfset * fGainFactor) ;
END_METHOD

END_FUNCTION_BLOCK

// Sensors/AnalogInput/FunctionBlocks/FB_DevHDAnalogInAutoCalibrate
FUNCTION_BLOCK PUBLIC FB_DevHDAnalogInAutoCalibrate EXTENDS FB_DevHDAnalogInputScaled
VAR_INPUT
END_VAR
VAR_OUTPUT
END_VAR
VAR
END_VAR

SUPER^();

METHOD PUBLIC CmdCalibrateNull : BOOL
VAR_INPUT
END_VAR
// set offset to calibrate to null
nOfset := - inHwInput ;
END_METHOD

METHOD PUBLIC CmdCalilbrateValue : BOOL // calibrate gain factor to actual value (warning calibrate to null before calibrating to value)
VAR_INPUT
	fCalibrationValue	: LREAL ; // Active input value to sensor (calibration setpoint)
END_VAR
// set gain from current value
fGainFactor := DINT_TO_LREAL(inHwInput + nOfset) / fCalibrationValue ;
END_METHOD

END_FUNCTION_BLOCK

// Sensors/AnalogInput/FunctionBlocks/FB_DevHDAnalogInputScaled
FUNCTION_BLOCK PUBLIC FB_DevHDAnalogInputScaled EXTENDS FB_DevHDAnalogInput
VAR_INPUT
END_VAR
VAR_OUTPUT
END_VAR
VAR
	fGainFactor 	: LREAL	:= 1	;
	nOfset			: DINT	:= 0	;
END_VAR

SUPER^();

METHOD ExecSetFeedback : BOOL
VAR
	nCalibValue	: DINT ; 
END_VAR
// Offset 
IF bCmdSimulate THEN 
	nCalibValue := fSimValue + nOfset ;
ELSE
	nCalibValue := inHwInput + nOfset ;
END_IF

fValue := DINT_TO_LREAL(nCalibValue) / fGainFactor;
END_METHOD

METHOD PUBLIC SetScaling : BOOL 
VAR_INPUT
	fMaxValue	: LREAL ; 	// Maximum input value after scaling, e.g. 100%, 0 = no scaling (gain = hardware limit / fMaxValue)  
	fOfset		: LREAL ;	// offset value (fvalue = (gain * hwvalue) + fOfset)
END_VAR
// calculate gain 
IF fMaxValue =0 THEN 
	fGainFactor := 1 ;
ELSE 
	fGainFactor := nLimitMax / fMaxValue ;
END_IF

nOfset := LREAL_TO_DINT(fOfset * fGainFactor) ;

SetScaling := TRUE ;
END_METHOD

END_FUNCTION_BLOCK

// Sensors/AnalogInput/FunctionBlocks/FB_DevHDAnalogInput
FUNCTION_BLOCK PUBLIC FB_DevHDAnalogInput EXTENDS FB_DevBase
VAR_INPUT
	bCmdSimulate	: BOOL 	:= FALSE ;// Simulate sensor Input 
	fSimValue		: DINT	:= 0 ;// Simulated sensor state
END_VAR
VAR_OUTPUT
	fValue	: LREAL := 0 ; // Analog input value (LREAL)
END_VAR
VAR
	nLimitMin		: DINT := Utilities_Library.GVL_FixedValues.nDINTMINVALUE	; // Initial value is set to integer minimum value for use with normal def analog inputs 
	nLimitMax 		: DINT := Utilities_Library.GVL_FixedValues.nDINTMAXVALUE 	; // Initial value is set to integer minimum value for use with high def analog inputs
	inHwInput AT%I* : DINT ; // Hardware connection
END_VAR

// Set device type
eDevType := E_Devices.AnalogSensor ;

// Call base function
SUPER^();

// set feedback
ExecSetFeedback();

METHOD ExecSetFeedback : BOOL
VAR_INPUT
END_VAR
IF bCmdSimulate THEN 
	fValue := fSimValue ;
ELSE
	fValue := DINT_TO_LREAL(inHwInput);
END_IF
END_METHOD

END_FUNCTION_BLOCK

// Sensors/FootPedals/FunctionBlocks/FB_EfkaEB301A_FootPedal
FUNCTION_BLOCK PUBLIC FB_EfkaEB301A_FootPedal
VAR_INPUT
	bEnable : BOOL := TRUE ;
END_VAR
VAR_OUTPUT
	ePedalInputStep		: E_FootpedalPos	:= 0 ;
	bRTrigtoReverse1 	: BOOL := FALSE ; // rising edge trigger when pedal moves from 0 to -1 or Idle to reverse 1 
	bRTrigtoReverse2 	: BOOL := FALSE ; // rising edge trigger when pedal moves from 1 to -2 or reverse 1 to reverse 2 
	bRTrigtoForward1 	: BOOL := FALSE ; // rising edge trigger when pedal moves from 0 to 1 or idle to forward 1 
	bRTrigtoForward2 	: BOOL := FALSE ; // rising edge trigger when pedal moves from 0 to 1 or forward to forward 2 
END_VAR
VAR
	// ===== greycode switches from footpedal =====
	I_GreyCodeA AT%I* : BOOL	; // Greycode input a from foot pedal 
	I_GreyCodeB AT%I* : BOOL	; // Greycode input a from foot pedal 
	I_GreyCodeC AT%I* : BOOL	; // Greycode input a from foot pedal 
	I_GreyCodeD AT%I* : BOOL	; // Greycode input a from foot pedal 
	nGreyCodetotal	: BYTE ; // all greycode switches combined
	// ==== decimal value =====
	ePreviousPedalInput	: E_FootpedalPos	:= 0 ;
END_VAR

// ===== Read input from pedal =====
ACT_ConvertGreycode();

// ===== Create edge flanks for functions =====
ACT_CreateEdges();

ACTION ACT_ConvertGreycode:
// ===== Combine greycode sensors =====
nGreyCodetotal.0 := I_GreyCodeA ;
nGreyCodetotal.1 := I_GreyCodeB ;
nGreyCodetotal.2 := I_GreyCodeB ;
nGreyCodetotal.3 := I_GreyCodeC ;

// ==== Convert greycode decimal to speed steps =====
// this only makes sense in EFKA world but anyway let's convert it to our own sense
CASE nGreyCodetotal OF 
	12: ePedalInputStep := E_FootpedalPos.eReverse1	;
	14: ePedalInputStep := E_FootpedalPos.eReverse2	;
	15: ePedalInputStep := E_FootpedalPos.eIdle		;
	13: ePedalInputStep := E_FootpedalPos.eForward1	;
	09: ePedalInputStep := E_FootpedalPos.eForward2	;
 	08: ePedalInputStep := E_FootpedalPos.eForward3	;
	10: ePedalInputStep := E_FootpedalPos.eForward4	;
	11: ePedalInputStep := E_FootpedalPos.eForward5	;
	03:	ePedalInputStep := E_FootpedalPos.eForward6	;
	02:	ePedalInputStep := E_FootpedalPos.eForward7	;
	00: ePedalInputStep := E_FootpedalPos.eForward8	;
	01: ePedalInputStep := E_FootpedalPos.eForward9	;
	05: ePedalInputStep := E_FootpedalPos.eForward10	;
	04: ePedalInputStep := E_FootpedalPos.eForward11	;
	06: ePedalInputStep := E_FootpedalPos.eForward12 	;
	07: ePedalInputStep := E_FootpedalPos.eForward13	;
	ELSE
		ePedalInputStep := E_FootpedalPos.eFalse 		;
END_CASE
END_ACTION

ACTION ACT_CreateEdges:
// ===== create edges on which functions can be triggerd =====
CASE ePedalInputStep OF
	E_FootpedalPos.eReverse2:
		bRTrigtoReverse2 := ePreviousPedalInput = E_FootpedalPos.eReverse1 ;
	E_FootpedalPos.eReverse1:
		bRTrigtoReverse1 := ePreviousPedalInput = E_FootpedalPos.eIdle ;
	E_FootpedalPos.eForward1:
		bRTrigtoForward1 := ePreviousPedalInput = E_FootpedalPos.eIdle ;
	E_FootpedalPos.eForward2: 
		bRTrigtoForward2 := ePreviousPedalInput = E_FootpedalPos.eForward1 ; 
END_CASE 

// write previous pedal input 
ePreviousPedalInput := ePedalInputStep ;
END_ACTION

END_FUNCTION_BLOCK

// Sensors/ModuleSpecific/EL3556_Loadcell/Fb_DevEL3356_LoadCell
FUNCTION_BLOCK PUBLIC Fb_DevEL3356_LoadCell EXTENDS FB_DevHDAnalogInAutoCalibrate
VAR_INPUT
	tCalibrationDelay	: TIME := T#2S ; // Time for which the load neads to before calibration is done (default T#2s) 
END_VAR
VAR_OUTPUT
	bMeasurementError	: BOOL 		; // Measurement or component error is active
	sErroDiscription 	: STRING 	; // 
END_VAR
VAR
	ibOverrange				AT%I*	: BOOL ; // overrange status indication
	ibDataInvalid			AT%I*	: BOOL ; // Data is invalid
	ibError					AT%I*	: BOOL ; // Module is in error state
	ibCalibrationinProgress	AT%I*	: BOOL ; // automatic calibration is in progress
	ibSteadyState			AT%I*	: BOOL ; // Module is in steady state
	ibSyncError				AT%I*	: BOOL ; // Module sync error
	
	tonSteadyState	: TON ; // steady state delay for calibration
END_VAR

ACTION CheckELSignalState:
// Set error device measurement error bit
bMeasurementError := FALSE ;

IF ibOverrange THEN 
	bMeasurementError 	S= TRUE;
 	sErroDiscription	:= 'Load exceeds maximum range ';
ELSIF ibDataInvalid THEN
	bMeasurementError 	S= TRUE;
	sErroDiscription	:= 'Incorrect date from device';
ELSIF ibError THEN
	bMeasurementError 	S= TRUE;
	sErroDiscription	:= 'Module general error';
ELSIF ibCalibrationinProgress THEN
	bMeasurementError 	S= TRUE;
	sErroDiscription	:= 'Calibration session in progress';
ELSIF ibSyncError THEN
	bMeasurementError 	S= TRUE;
	sErroDiscription	:= 'Module ethercat sync error';	
END_IF
END_ACTION

METHOD PUBLIC CmdCalibrateNull : BOOL
VAR_INPUT
END_VAR
tonSteadyState(IN := ibSteadyState, PT := tCalibrationDelay);

// set offset to calibrate to null
IF tonSteadyState.Q THEN 
	nOfset := - inHwInput ;
END_IF
END_METHOD

METHOD PUBLIC CmdCalilbrateValue : BOOL // calibrate gain factor to actual value (warning calibrate to null before calibrating to value)
VAR_INPUT
	fCalibrationValue	: LREAL ; // Active input value to sensor [N]
END_VAR
tonSteadyState(IN := ibSteadyState, PT := tCalibrationDelay);

// set gain from current value
IF tonSteadyState.Q THEN 
	fGainFactor := DINT_TO_LREAL(inHwInput + nOfset) / fCalibrationValue ; 
END_IF
END_METHOD

END_FUNCTION_BLOCK
